{attribute 'qualified_only'}
VAR_GLOBAL CONSTANT
	MaxAmountProgramChildren				: UINT := 10;
END_VAR

(* stored: Version 1.1.0.1
   GVL Par_Core: Id {af0443aa-dedc-4249-a29a-4ebfacc13643}, ParameterList True *)
